{attribute 'qualified_only'}
{attribute 'strict'}
{attribute 'to_string'}
TYPE AUTOMATION_ENGINE_STATE :
(
	INITIALIZING := 0, // It acts until at least one unit has not completed initialization
    RUNNING := 1, // Normal running            
	EMERGENCY := 2,	// Emergency stop initiated
    FAULT := 3 // Any error occurred while initializing or fatal error in other modes
);
END_TYPE

(* stored: Version 1.1.0.1
   DUT AUTOMATION_ENGINE_STATE: Id {e0aa6b66-b856-4339-85da-3620262659fe} *)
